SUBAPPLICATION Uebung_025 (* Spiegelabfolge (5) *)
  (* Standard: 61499-2; Description: Copyright (c) 2023 Meisterschulen am Ostbahnhof This program and the accompanying materials are made available under the terms of the Eclipse Public License 2.0 which is available at https://www.eclipse.org/legal/epl-2.0/ SPDX-License-Identifier: EPL-2.0 *)
  (* Version 1.0, 2023-10-23, Franz Höpfinger, Meisterschulen am Ostbahnhof *)
  IMPORT logiBUS::io::DI::logiBUS_DI;
  IMPORT logiBUS::io::DQ::logiBUS_DO;
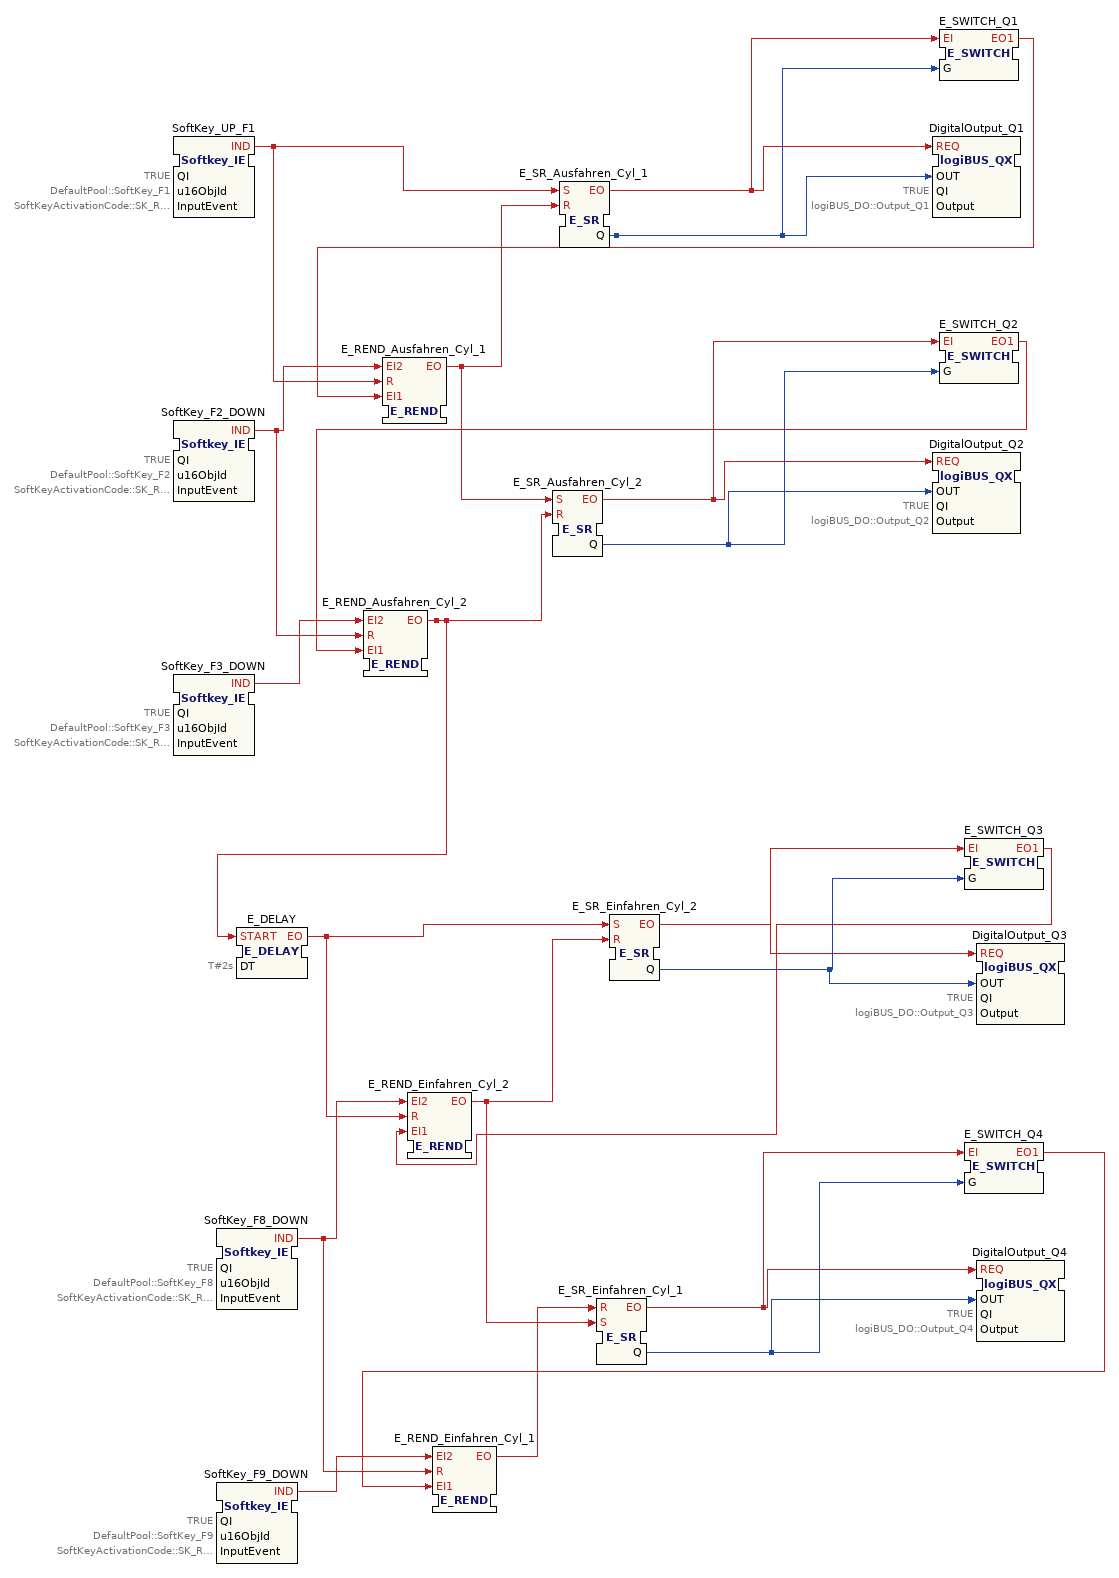
  (* START-Knopf Ausfahren *)
  (* Endlage Ausfahren_Cyl_1 *)
  (* Endlage Ausfahren_Cyl_2 *)
  (* Ausfahren_Cyl_1 *)
  (* Ausfahren_Cyl_2 *)
  (* Einfahren Zeit gesteuert *)
  (* Endlage Einfahren_Cyl_1 *)
  (* Einfahren_Cyl_2 *)
  (* Endlage Einfahren_Cyl_2 *)
  (* Einfahren_Cyl_1 *)
  FBS
    DigitalOutput_Q1 : logiBUS::io::DQ::logiBUS_QX(QI := TRUE, Output := logiBUS_DO::Output_Q1);
    SoftKey_UP_F1 : Softkey_IE(QI := TRUE, u16ObjId := DefaultPool::SoftKey_F1, InputEvent := SoftKeyActivationCode::SK_RELEASED);
    E_SR_Ausfahren_Cyl_1 : E_SR;
    SoftKey_F2_DOWN : Softkey_IE(QI := TRUE, u16ObjId := DefaultPool::SoftKey_F2, InputEvent := SoftKeyActivationCode::SK_RELEASED);
    DigitalOutput_Q2 : logiBUS::io::DQ::logiBUS_QX(QI := TRUE, Output := logiBUS_DO::Output_Q2);
    E_SR_Ausfahren_Cyl_2 : E_SR;
    SoftKey_F3_DOWN : Softkey_IE(QI := TRUE, u16ObjId := DefaultPool::SoftKey_F3, InputEvent := SoftKeyActivationCode::SK_RELEASED);
    SoftKey_F9_DOWN : Softkey_IE(QI := TRUE, u16ObjId := DefaultPool::SoftKey_F9, InputEvent := SoftKeyActivationCode::SK_RELEASED);
    E_SR_Einfahren_Cyl_2 : E_SR;
    DigitalOutput_Q3 : logiBUS::io::DQ::logiBUS_QX(QI := TRUE, Output := logiBUS_DO::Output_Q3);
    DigitalOutput_Q4 : logiBUS::io::DQ::logiBUS_QX(QI := TRUE, Output := logiBUS_DO::Output_Q4);
    E_SR_Einfahren_Cyl_1 : E_SR;
    SoftKey_F8_DOWN : Softkey_IE(QI := TRUE, u16ObjId := DefaultPool::SoftKey_F8, InputEvent := SoftKeyActivationCode::SK_RELEASED);
    E_DELAY : E_DELAY(DT := T#2s);
    E_REND_Ausfahren_Cyl_1 : E_REND;
    E_REND_Ausfahren_Cyl_2 : E_REND;
    E_REND_Einfahren_Cyl_2 : E_REND;
    E_REND_Einfahren_Cyl_1 : E_REND;
    E_SWITCH_Q1 : E_SWITCH;
    E_SWITCH_Q2 : E_SWITCH;
    E_SWITCH_Q3 : E_SWITCH;
    E_SWITCH_Q4 : E_SWITCH;
  END_FBS
  EVENT_CONNECTIONS
    SoftKey_UP_F1.IND TO E_SR_Ausfahren_Cyl_1.S;
    E_SR_Ausfahren_Cyl_1.EO TO DigitalOutput_Q1.REQ;
    E_SR_Ausfahren_Cyl_2.EO TO DigitalOutput_Q2.REQ;
    E_SR_Einfahren_Cyl_2.EO TO DigitalOutput_Q3.REQ;
    E_SR_Einfahren_Cyl_1.EO TO DigitalOutput_Q4.REQ;
    E_DELAY.EO TO E_SR_Einfahren_Cyl_2.S;
    E_REND_Ausfahren_Cyl_1.EO TO E_SR_Ausfahren_Cyl_1.R;
    E_REND_Ausfahren_Cyl_1.EO TO E_SR_Ausfahren_Cyl_2.S;
    SoftKey_F2_DOWN.IND TO E_REND_Ausfahren_Cyl_1.EI2;
    SoftKey_F3_DOWN.IND TO E_REND_Ausfahren_Cyl_2.EI2;
    E_REND_Ausfahren_Cyl_2.EO TO E_SR_Ausfahren_Cyl_2.R;
    E_REND_Einfahren_Cyl_1.EO TO E_SR_Einfahren_Cyl_1.R;
    SoftKey_F9_DOWN.IND TO E_REND_Einfahren_Cyl_1.EI2;
    E_REND_Einfahren_Cyl_2.EO TO E_SR_Einfahren_Cyl_1.S;
    E_REND_Einfahren_Cyl_2.EO TO E_SR_Einfahren_Cyl_2.R;
    SoftKey_F8_DOWN.IND TO E_REND_Einfahren_Cyl_2.EI2;
    E_REND_Ausfahren_Cyl_2.EO TO E_DELAY.START;
    SoftKey_UP_F1.IND TO E_REND_Ausfahren_Cyl_1.R;
    SoftKey_F2_DOWN.IND TO E_REND_Ausfahren_Cyl_2.R;
    E_DELAY.EO TO E_REND_Einfahren_Cyl_2.R;
    SoftKey_F8_DOWN.IND TO E_REND_Einfahren_Cyl_1.R;
    E_SR_Einfahren_Cyl_1.EO TO E_SWITCH_Q4.EI;
    E_SR_Einfahren_Cyl_2.EO TO E_SWITCH_Q3.EI;
    E_SR_Ausfahren_Cyl_2.EO TO E_SWITCH_Q2.EI;
    E_SR_Ausfahren_Cyl_1.EO TO E_SWITCH_Q1.EI;
    E_SWITCH_Q1.EO1 TO E_REND_Ausfahren_Cyl_1.EI1;
    E_SWITCH_Q2.EO1 TO E_REND_Ausfahren_Cyl_2.EI1;
    E_SWITCH_Q3.EO1 TO E_REND_Einfahren_Cyl_2.EI1;
    E_SWITCH_Q4.EO1 TO E_REND_Einfahren_Cyl_1.EI1;
  END_CONNECTIONS
  DATA_CONNECTIONS
    E_SR_Ausfahren_Cyl_1.Q TO DigitalOutput_Q1.OUT;
    E_SR_Ausfahren_Cyl_2.Q TO DigitalOutput_Q2.OUT;
    E_SR_Einfahren_Cyl_1.Q TO DigitalOutput_Q4.OUT;
    E_SR_Einfahren_Cyl_2.Q TO DigitalOutput_Q3.OUT;
    E_SR_Einfahren_Cyl_1.Q TO E_SWITCH_Q4.G;
    E_SR_Einfahren_Cyl_2.Q TO E_SWITCH_Q3.G;
    E_SR_Ausfahren_Cyl_2.Q TO E_SWITCH_Q2.G;
    E_SR_Ausfahren_Cyl_1.Q TO E_SWITCH_Q1.G;
  END_CONNECTIONS
END_SUBAPPLICATION
